// TIA Portal project "PLC_5a_DF_2024compl_V17" (V17)

(* hardware
DEVICE "S7-1200 station_1"  S7-1200 Station
   slot 0: "Telaio di montaggio_0"  S7-1200 Rack  Rack  V1.0
   slot 1: "PLC_ImpiantoCarta"  CPU 1215C DC/DC/Rly  6ES7 215-1HG40-0XB0  V4.5
DEVICE "HMI_1"  TP700 Comfort
   slot 0: "HMI_1"  TP700 Comfort  6AV2 124-0GC01-0AX0  17.0.0.0
   slot 1: "HMI_RT_1"  TP700 Comfort  6AV2 124-0GC01-0AX0  17.0.0.0
   slot 5: "HMI_1.IE_CP_1"  PROFINET Interface  17.0.0.0
      slot 1: "Interfaccia_1 PROFINET"  PROFINET Interface
         slot 1: "Porta_1"  Port
         slot 2: "Porta_2"  Port
   slot 7: "HMI_1.MPI/DP_CP_1"  MPI/DP Interface  17.0.0.0
*)

// ===== PLC "PLC_ImpiantoCarta"  CPU 1215C DC/DC/Rly =====

VAR_GLOBAL   // PLC tag table "Tabella delle variabili standard"
   "M_all_Ms" AT %M10.0 : Bool;   // Memoria allarme Ms
   "M_all_Mn" AT %M10.1 : Bool;   // Memoria allarme Mn
   "M_all_Mp" AT %M10.2 : Bool;   // Memoria allarme Mp
   "M_all_Yv" AT %M10.3 : Bool;   // Memoria allarme Yv
   "Ciclo_Auto" AT %M20.0 : Bool;   // Ciclo automatico
   "Riempimento" AT %M20.1 : Bool;   // Fase 1 di riempimento
   "Caricamento" AT %M20.2 : Bool;   // Fase 2
   "Miscelazione" AT %M20.3 : Bool;   // Fase 3
   "Attesa" AT %M20.4 : Bool;   // Fase 4
   "Svuotamento" AT %M20.5 : Bool;   // Fase 5
   "FN_S4" AT %M40.0 : Bool;   // Fronte discesa S4
   "System_Byte" AT %MB1 : Byte;
   "FirstScan" AT %M1.0 : Bool;
   "DiagStatusUpdate" AT %M1.1 : Bool;
   "AlwaysTRUE" AT %M1.2 : Bool;
   "AlwaysFALSE" AT %M1.3 : Bool;
   "Clock_Byte" AT %MB0 : Byte;
   "Clock_10Hz" AT %M0.0 : Bool;
   "Clock_5Hz" AT %M0.1 : Bool;
   "Clock_2.5Hz" AT %M0.2 : Bool;
   "Clock_2Hz" AT %M0.3 : Bool;
   "Clock_1.25Hz" AT %M0.4 : Bool;
   "Clock_1Hz" AT %M0.5 : Bool;
   "Clock_0.625Hz" AT %M0.6 : Bool;
   "Clock_0.5Hz" AT %M0.7 : Bool;
END_VAR

VAR_GLOBAL   // PLC tag table "IO"
   "S1" AT %I0.0 : Bool;   // Sensore di minimo livello
   "S2" AT %I0.1 : Bool;   // Sensore livello lavoro
   "S3" AT %I0.2 : Bool;   // Sensore di massimo livello
   "S4" AT %I0.3 : Bool;   // Sensore conteggio pezzi
   "Term_Ms" AT %I0.4 : Bool;   // Termico motore Ms (1=OK)
   "Term_Mn" AT %I0.5 : Bool;   // Termico motore Mn (1=OK)
   "Term_Mp" AT %I0.6 : Bool;   // Termico motore Mp (1=OK)
   "YvMicrO" AT %I0.7 : Bool;   // Sensore valvola Yv aperta
   "Motor_Ms" AT %Q0.0 : Bool;   // Motore spappolatore
   "Motor_Mn" AT %Q0.1 : Bool;   // Motore nastro
   "Motor_Mp" AT %Q0.2 : Bool;   // Pompa svuotamento
   "Yv" AT %Q0.3 : Bool;   // Valvola riempimento
   "H1" AT %Q0.4 : Bool;   // Lampada attesa per svuotamento
   "Hs" AT %Q0.5 : Bool;   // Lampada Ms
   "Hn" AT %Q0.6 : Bool;   // Lampada Mn
   "Hp" AT %Q0.7 : Bool;   // Lampada Mp
   "Hv" AT %Q1.0 : Bool;   // Lampada Yv
END_VAR

DATA_BLOCK "DB_HMI"   // DB1
{ S7_Optimized_Access := 'TRUE' }
VERSION : 0.1
   VAR
      SEL_ManAut : Bool;   // SELETTORE DI FUNZIONAMENTO (1=auto)
      Sa : Bool;   // PULSANTE DI START CICLO
      Sp : Bool;   // PULSANTE SVUOTAMENTO
      St : Bool;   // PULSANTE DI STOP CICLO
      Reset : Bool;   // RESET ALLARMI
      CMD_MAN : Struct
         Ms_Start : Bool;   // COMANDO MANUALE START Ms
         Ms_Stop : Bool;   // COMANDO MANUALE ARRESTO Ms
         Mn_Start : Bool;   // COMANDO MANUALE START Mn
         Mn_Stop : Bool;   // COMANDO MANUALE ARRESTO Mn
         Mp_Start : Bool;   // COMANDO MANUALE START Mp
         Mp_Stop : Bool;   // COMANDO MANUALE ARRESTO Mp
         Yv_On : Bool;   // COMANDO MANUALE ECCITA Yv
         Yv_Off : Bool;   // COMANDO MANUALE DISECCITA Yv
      END_STRUCT;
   END_VAR
   VAR RETAIN
      Param : Struct
         PT_Timeout_Yv : Time := T#3s;   // Timeout apertura valvola
         Num_pezzi_da_caricare : Int := 10;   // Numero pezzi da caricare
         Num_pezzi_contati : Int;   // Numero pezzi contati
         Tempo_Miscelazione : Time := T#20S;   // Tempo miscelazione
      END_STRUCT;
   END_VAR
BEGIN
END_DATA_BLOCK

// folder: System blocks/Program resources

DATA_BLOCK "RIT_ALL_Yv"   // DB2
{ S7_Optimized_Access := 'TRUE' }
AUTHOR : Simatic
FAMILY : IEC
NAME : IEC_TMR
VERSION : 1.0
// stored: InstanceOfName IEC_TIMER
"IEC_TIMER"
BEGIN
END_DATA_BLOCK

DATA_BLOCK "DB_Miscelazione"   // DB3
{ S7_Optimized_Access := 'TRUE' }
AUTHOR : Simatic
FAMILY : IEC
NAME : IEC_TMR
VERSION : 1.0
// stored: InstanceOfName IEC_TIMER
"IEC_TIMER"
BEGIN
END_DATA_BLOCK

// folder: (top level)

FUNCTION "DISPOSITIVI" : Void   // FC1, LAD
TITLE = Gestione motori e valvola
{ S7_Optimized_Access := 'TRUE' }
VERSION : 0.1
BEGIN

REGION Network 1: Valvola riempimento
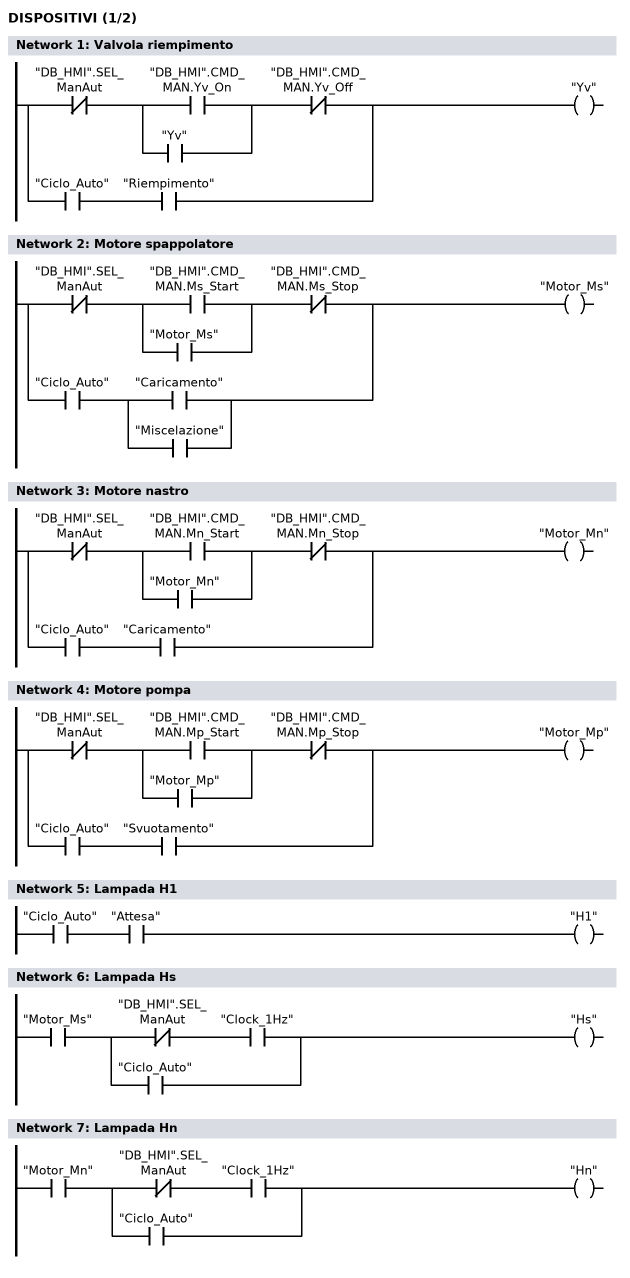
   RUNG wire#powerrail
      I_Contact( "DB_HMI".SEL_ManAut )
      wire#w1
      Contact( "DB_HMI".CMD_MAN.Yv_On )
      wire#w2
      I_Contact( "DB_HMI".CMD_MAN.Yv_Off )
      wire#w3
      Coil( "Yv" )
   END_RUNG
   RUNG wire#w1
      Contact( "Yv" )
   END_RUNG wire#w2
   RUNG wire#powerrail
      Contact( "Ciclo_Auto" )
      Contact( "Riempimento" )
   END_RUNG wire#w3
   // the same network as SCL:
   "Yv" := (NOT "DB_HMI".SEL_ManAut AND ("DB_HMI".CMD_MAN.Yv_On OR "Yv") AND NOT "DB_HMI".CMD_MAN.Yv_Off) OR ("Ciclo_Auto" AND "Riempimento");
END_REGION

REGION Network 2: Motore spappolatore
   RUNG wire#powerrail
      I_Contact( "DB_HMI".SEL_ManAut )
      wire#w1
      Contact( "DB_HMI".CMD_MAN.Ms_Start )
      wire#w2
      I_Contact( "DB_HMI".CMD_MAN.Ms_Stop )
      wire#w3
      Coil( "Motor_Ms" )
   END_RUNG
   RUNG wire#w1
      Contact( "Motor_Ms" )
   END_RUNG wire#w2
   RUNG wire#powerrail
      Contact( "Ciclo_Auto" )
      wire#w4
      Contact( "Caricamento" )
   END_RUNG wire#w3
   RUNG wire#w4
      Contact( "Miscelazione" )
   END_RUNG wire#w3
   // the same network as SCL:
   "Motor_Ms" := (NOT "DB_HMI".SEL_ManAut AND ("DB_HMI".CMD_MAN.Ms_Start OR "Motor_Ms") AND NOT "DB_HMI".CMD_MAN.Ms_Stop) OR ("Ciclo_Auto" AND ("Caricamento" OR "Miscelazione"));
END_REGION

REGION Network 3: Motore nastro
   RUNG wire#powerrail
      I_Contact( "DB_HMI".SEL_ManAut )
      wire#w1
      Contact( "DB_HMI".CMD_MAN.Mn_Start )
      wire#w2
      I_Contact( "DB_HMI".CMD_MAN.Mn_Stop )
      wire#w3
      Coil( "Motor_Mn" )
   END_RUNG
   RUNG wire#w1
      Contact( "Motor_Mn" )
   END_RUNG wire#w2
   RUNG wire#powerrail
      Contact( "Ciclo_Auto" )
      Contact( "Caricamento" )
   END_RUNG wire#w3
   // the same network as SCL:
   "Motor_Mn" := (NOT "DB_HMI".SEL_ManAut AND ("DB_HMI".CMD_MAN.Mn_Start OR "Motor_Mn") AND NOT "DB_HMI".CMD_MAN.Mn_Stop) OR ("Ciclo_Auto" AND "Caricamento");
END_REGION

REGION Network 4: Motore pompa
   RUNG wire#powerrail
      I_Contact( "DB_HMI".SEL_ManAut )
      wire#w1
      Contact( "DB_HMI".CMD_MAN.Mp_Start )
      wire#w2
      I_Contact( "DB_HMI".CMD_MAN.Mp_Stop )
      wire#w3
      Coil( "Motor_Mp" )
   END_RUNG
   RUNG wire#w1
      Contact( "Motor_Mp" )
   END_RUNG wire#w2
   RUNG wire#powerrail
      Contact( "Ciclo_Auto" )
      Contact( "Svuotamento" )
   END_RUNG wire#w3
   // the same network as SCL:
   "Motor_Mp" := (NOT "DB_HMI".SEL_ManAut AND ("DB_HMI".CMD_MAN.Mp_Start OR "Motor_Mp") AND NOT "DB_HMI".CMD_MAN.Mp_Stop) OR ("Ciclo_Auto" AND "Svuotamento");
END_REGION

REGION Network 5: Lampada H1
   RUNG wire#powerrail
      Contact( "Ciclo_Auto" )
      Contact( "Attesa" )
      Coil( "H1" )
   END_RUNG
   // the same network as SCL:
   "H1" := "Ciclo_Auto" AND "Attesa";
END_REGION

REGION Network 6: Lampada Hs
   RUNG wire#powerrail
      Contact( "Motor_Ms" )
      wire#w1
      I_Contact( "DB_HMI".SEL_ManAut )
      Contact( "Clock_1Hz" )
      wire#w2
      Coil( "Hs" )
   END_RUNG
   RUNG wire#w1
      Contact( "Ciclo_Auto" )
   END_RUNG wire#w2
   // the same network as SCL:
   "Hs" := "Motor_Ms" AND ((NOT "DB_HMI".SEL_ManAut AND "Clock_1Hz") OR "Ciclo_Auto");
END_REGION

REGION Network 7: Lampada Hn
   RUNG wire#powerrail
      Contact( "Motor_Mn" )
      wire#w1
      I_Contact( "DB_HMI".SEL_ManAut )
      Contact( "Clock_1Hz" )
      wire#w2
      Coil( "Hn" )
   END_RUNG
   RUNG wire#w1
      Contact( "Ciclo_Auto" )
   END_RUNG wire#w2
   // the same network as SCL:
   "Hn" := "Motor_Mn" AND ((NOT "DB_HMI".SEL_ManAut AND "Clock_1Hz") OR "Ciclo_Auto");
END_REGION

REGION Network 8: Lampada Hp
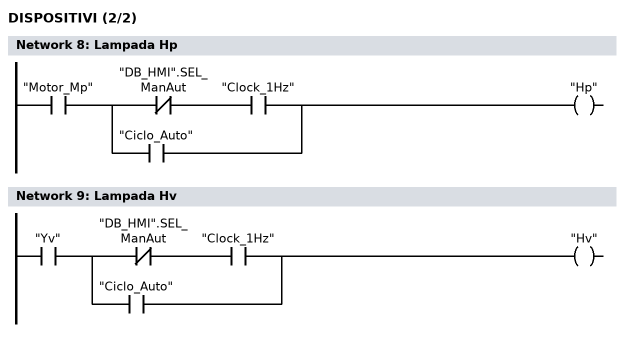
   RUNG wire#powerrail
      Contact( "Motor_Mp" )
      wire#w1
      I_Contact( "DB_HMI".SEL_ManAut )
      Contact( "Clock_1Hz" )
      wire#w2
      Coil( "Hp" )
   END_RUNG
   RUNG wire#w1
      Contact( "Ciclo_Auto" )
   END_RUNG wire#w2
   // the same network as SCL:
   "Hp" := "Motor_Mp" AND ((NOT "DB_HMI".SEL_ManAut AND "Clock_1Hz") OR "Ciclo_Auto");
END_REGION

REGION Network 9: Lampada Hv
   RUNG wire#powerrail
      Contact( "Yv" )
      wire#w1
      I_Contact( "DB_HMI".SEL_ManAut )
      Contact( "Clock_1Hz" )
      wire#w2
      Coil( "Hv" )
   END_RUNG
   RUNG wire#w1
      Contact( "Ciclo_Auto" )
   END_RUNG wire#w2
   // the same network as SCL:
   "Hv" := "Yv" AND ((NOT "DB_HMI".SEL_ManAut AND "Clock_1Hz") OR "Ciclo_Auto");
END_REGION
END_FUNCTION

FUNCTION "ALLARMI" : Void   // FC2, LAD
{ S7_Optimized_Access := 'TRUE' }
VERSION : 0.1
BEGIN

REGION Network 1: ALLARME MOTORE Ms
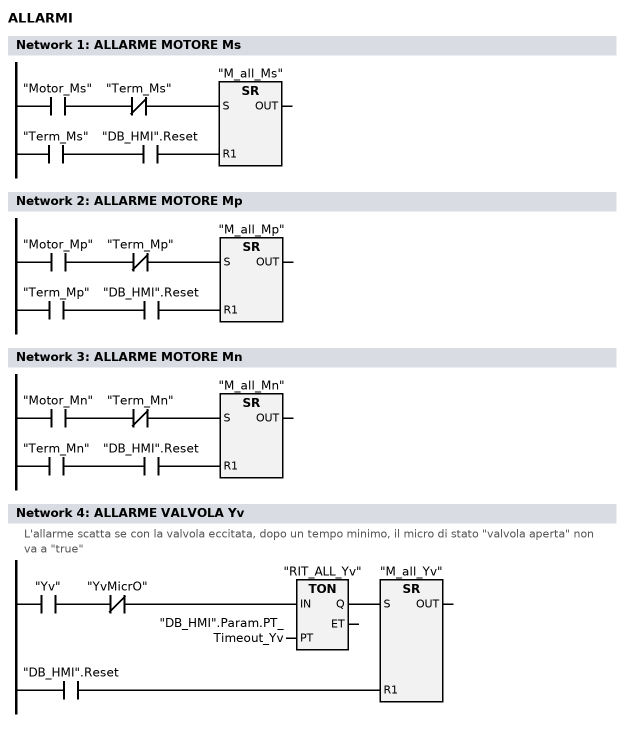
   RUNG wire#powerrail
      Contact( "Motor_Ms" )
      I_Contact( "Term_Ms" )
      S_SR(operand := "M_all_Ms", r1 := wire#w1)
   END_RUNG
   RUNG wire#powerrail
      Contact( "Term_Ms" )
      Contact( "DB_HMI".Reset )
   END_RUNG wire#w1
   // the same network as SCL:
   IF "Motor_Ms" AND NOT "Term_Ms" THEN
       "M_all_Ms" := TRUE;   // SR flip-flop
   END_IF;
   IF "Term_Ms" AND "DB_HMI".Reset THEN "M_all_Ms" := FALSE; END_IF;
END_REGION

REGION Network 2: ALLARME MOTORE Mp
   RUNG wire#powerrail
      Contact( "Motor_Mp" )
      I_Contact( "Term_Mp" )
      S_SR(operand := "M_all_Mp", r1 := wire#w1)
   END_RUNG
   RUNG wire#powerrail
      Contact( "Term_Mp" )
      Contact( "DB_HMI".Reset )
   END_RUNG wire#w1
   // the same network as SCL:
   IF "Motor_Mp" AND NOT "Term_Mp" THEN
       "M_all_Mp" := TRUE;   // SR flip-flop
   END_IF;
   IF "Term_Mp" AND "DB_HMI".Reset THEN "M_all_Mp" := FALSE; END_IF;
END_REGION

REGION Network 3: ALLARME MOTORE Mn
   RUNG wire#powerrail
      Contact( "Motor_Mn" )
      I_Contact( "Term_Mn" )
      S_SR(operand := "M_all_Mn", r1 := wire#w1)
   END_RUNG
   RUNG wire#powerrail
      Contact( "Term_Mn" )
      Contact( "DB_HMI".Reset )
   END_RUNG wire#w1
   // the same network as SCL:
   IF "Motor_Mn" AND NOT "Term_Mn" THEN
       "M_all_Mn" := TRUE;   // SR flip-flop
   END_IF;
   IF "Term_Mn" AND "DB_HMI".Reset THEN "M_all_Mn" := FALSE; END_IF;
END_REGION

REGION Network 4: ALLARME VALVOLA Yv
   // L'allarme scatta se con la valvola eccitata, dopo un tempo minimo, il micro di stato "valvola aperta" non va a "true"
   "RIT_ALL_Yv".TON(IN := "Yv" AND NOT "YvMicrO", PT := "DB_HMI".Param.PT_Timeout_Yv);
   IF "RIT_ALL_Yv".Q THEN
       "M_all_Yv" := TRUE;   // SR flip-flop
   END_IF;
   IF "DB_HMI".Reset THEN "M_all_Yv" := FALSE; END_IF;
END_REGION
END_FUNCTION

FUNCTION "CICLO_AUTOMATICO" : Void   // FC3, LAD
{ S7_Optimized_Access := 'TRUE' }
VERSION : 0.1
   VAR_TEMP   // added for the SCL form of the ladder/FBD networks
      _w1 : Bool;
   END_VAR
BEGIN

REGION Network 1: STOP CICLO (MOMENTANEO)
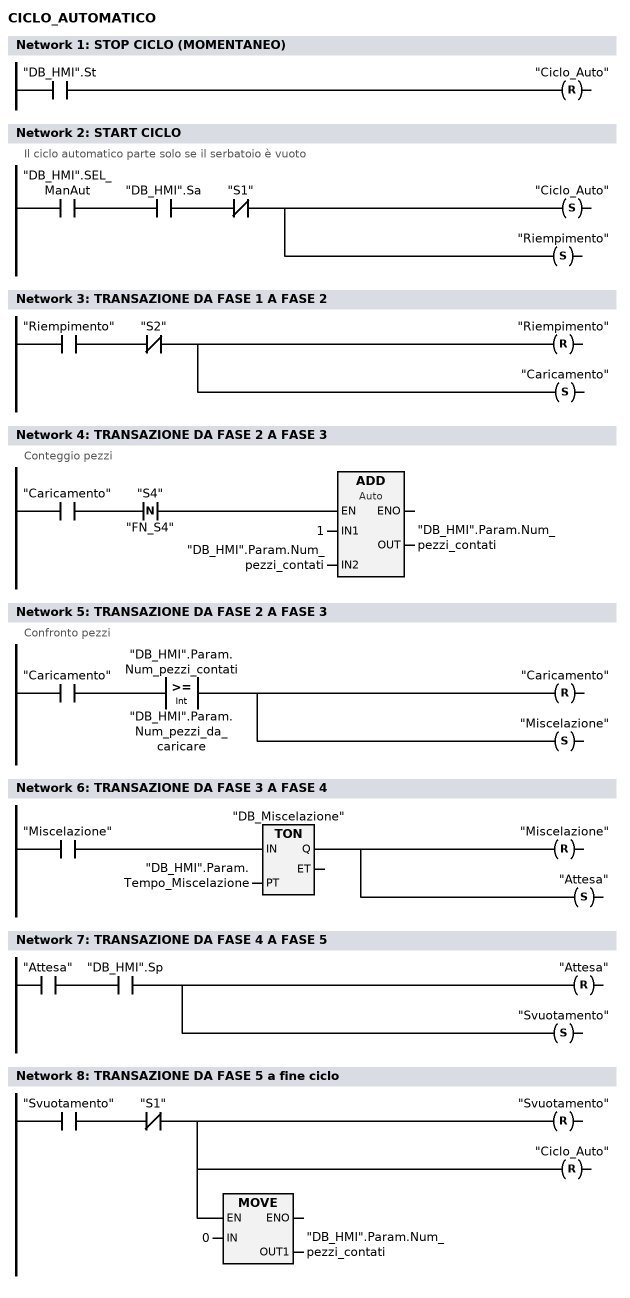
   RUNG wire#powerrail
      Contact( "DB_HMI".St )
      R_Coil( "Ciclo_Auto" )
   END_RUNG
   // the same network as SCL:
   IF "DB_HMI".St THEN "Ciclo_Auto" := FALSE; END_IF;
END_REGION

REGION Network 2: START CICLO
   // Il ciclo automatico parte solo se il serbatoio è vuoto
   RUNG wire#powerrail
      Contact( "DB_HMI".SEL_ManAut )
      Contact( "DB_HMI".Sa )
      I_Contact( "S1" )
      wire#w1
      S_Coil( "Ciclo_Auto" )
   END_RUNG
   RUNG wire#w1
      S_Coil( "Riempimento" )
   END_RUNG
   // the same network as SCL:
   IF "DB_HMI".SEL_ManAut AND "DB_HMI".Sa AND NOT "S1" THEN
       "Ciclo_Auto" := TRUE;
       "Riempimento" := TRUE;
   END_IF;
END_REGION

REGION Network 3: TRANSAZIONE DA FASE 1 A FASE 2
   RUNG wire#powerrail
      Contact( "Riempimento" )
      I_Contact( "S2" )
      wire#w1
      R_Coil( "Riempimento" )
   END_RUNG
   RUNG wire#w1
      S_Coil( "Caricamento" )
   END_RUNG
   // the same network as SCL:
   #_w1 := "Riempimento" AND NOT "S2";
   IF #_w1 THEN
       "Riempimento" := FALSE;
       "Caricamento" := TRUE;
   END_IF;
END_REGION

REGION Network 4: TRANSAZIONE DA FASE 2 A FASE 3
   // Conteggio pezzi
   RUNG wire#powerrail
      Contact( "Caricamento" )
      N_Contact(operand := "S4", bit := "FN_S4")
      Add(in1 := 1, in2 := "DB_HMI".Param.Num_pezzi_contati, out => "DB_HMI".Param.Num_pezzi_contati)
   END_RUNG
   // the same network as SCL:
   #_w1 := "Caricamento" AND NOT "S4" AND "FN_S4";   // falling edge of "S4"
   "FN_S4" := "S4";
   IF #_w1 THEN "DB_HMI".Param.Num_pezzi_contati := 1 + "DB_HMI".Param.Num_pezzi_contati; END_IF;
END_REGION

REGION Network 5: TRANSAZIONE DA FASE 2 A FASE 3
   // Confronto pezzi
   RUNG wire#powerrail
      Contact( "Caricamento" )
      { S7_Templates := "SrcType := Int" } GE_Contact(in1 := "DB_HMI".Param.Num_pezzi_contati, in2 := "DB_HMI".Param.Num_pezzi_da_caricare)
      wire#w1
      R_Coil( "Caricamento" )
   END_RUNG
   RUNG wire#w1
      S_Coil( "Miscelazione" )
   END_RUNG
   // the same network as SCL:
   #_w1 := "Caricamento" AND ("DB_HMI".Param.Num_pezzi_contati >= "DB_HMI".Param.Num_pezzi_da_caricare);
   IF #_w1 THEN
       "Caricamento" := FALSE;
       "Miscelazione" := TRUE;
   END_IF;
END_REGION

REGION Network 6: TRANSAZIONE DA FASE 3 A FASE 4
   "DB_Miscelazione".TON(IN := "Miscelazione", PT := "DB_HMI".Param.Tempo_Miscelazione);
   IF "DB_Miscelazione".Q THEN
       "Miscelazione" := FALSE;
       "Attesa" := TRUE;
   END_IF;
END_REGION

REGION Network 7: TRANSAZIONE DA FASE 4 A FASE 5
   RUNG wire#powerrail
      Contact( "Attesa" )
      Contact( "DB_HMI".Sp )
      wire#w1
      R_Coil( "Attesa" )
   END_RUNG
   RUNG wire#w1
      S_Coil( "Svuotamento" )
   END_RUNG
   // the same network as SCL:
   #_w1 := "Attesa" AND "DB_HMI".Sp;
   IF #_w1 THEN
       "Attesa" := FALSE;
       "Svuotamento" := TRUE;
   END_IF;
END_REGION

REGION Network 8: TRANSAZIONE DA FASE 5 a fine ciclo
   RUNG wire#powerrail
      Contact( "Svuotamento" )
      I_Contact( "S1" )
      wire#w1
      R_Coil( "Svuotamento" )
   END_RUNG
   RUNG wire#w1
      R_Coil( "Ciclo_Auto" )
   END_RUNG
   RUNG wire#w1
      Move(in := 0, out1 => "DB_HMI".Param.Num_pezzi_contati)
   END_RUNG
   // the same network as SCL:
   #_w1 := "Svuotamento" AND NOT "S1";
   IF #_w1 THEN
       "Svuotamento" := FALSE;
       "Ciclo_Auto" := FALSE;
       "DB_HMI".Param.Num_pezzi_contati := 0;
   END_IF;
END_REGION
END_FUNCTION

ORGANIZATION_BLOCK "Main"   // OB1, LAD, ProgramCycle
TITLE = "Main Program Sweep (Cycle)"
{ S7_Optimized_Access := 'TRUE' }
VERSION : 0.1
   VAR_INPUT
      Initial_Call : Bool;   // Initial call of this OB
      Remanence : Bool;   // =True, if remanent data are available
   END_VAR
BEGIN

REGION Network 1
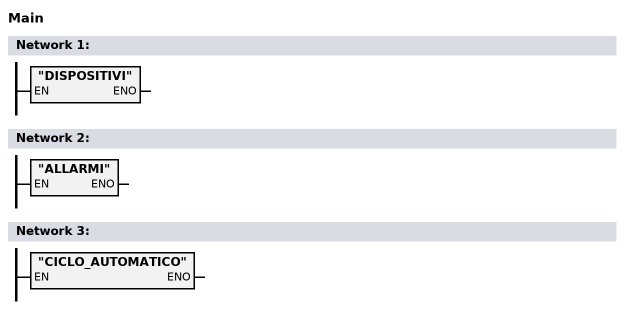
   RUNG wire#powerrail
      "DISPOSITIVI"()
   END_RUNG
   // the same network as SCL:
   "DISPOSITIVI"();
END_REGION

REGION Network 2
   RUNG wire#powerrail
      "ALLARMI"()
   END_RUNG
   // the same network as SCL:
   "ALLARMI"();
END_REGION

REGION Network 3
   RUNG wire#powerrail
      "CICLO_AUTOMATICO"()
   END_RUNG
   // the same network as SCL:
   "CICLO_AUTOMATICO"();
END_REGION
END_ORGANIZATION_BLOCK

(* ===== HMI "HMI_RT_1" =====
system functions are stored by id; their names below are inferred from use
connection "HMI_Collegamento_2": ETHERNET, S7_1200_OMS

HMI tags "Tabella delle variabili standard"
   "S3" : Bool = PLC S3 AT %I0.2, 1 s
   "Ms" : Bool = PLC Motor_Ms AT %Q0.0, 1 s
   "Mp" : Bool = PLC Motor_Mp AT %Q0.2, 1 s
   "Mn" : Bool = PLC Motor_Mn AT %Q0.1, 1 s
   "S4" : Bool = PLC S4 AT %I0.3, 1 s
   "S1" : Bool = PLC S1 AT %I0.0, 1 s
   "S2" : Bool = PLC S2 AT %I0.1, 1 s
   "Ciclo_Auto" : Bool = PLC Ciclo_Auto AT %M20.0, 1 s
   "Sa" : Bool = PLC DB_HMI.Sa AT %I0.0, 1 s
   "DB_HMI_CMD_MAN_Mn_Start" : Bool = PLC DB_HMI.CMD_MAN.Mn_Start, 1 s
   "DB_HMI_CMD_MAN_Mn_Stop" : Bool = PLC DB_HMI.CMD_MAN.Mn_Stop, 1 s
   "DB_HMI_Sp" : Bool = PLC DB_HMI.Sp, 1 s
   "DB_HMI_Sa" : Bool = PLC DB_HMI.Sa, 1 s
   "DB_HMI_SEL_ManAut" : Bool = PLC DB_HMI.SEL_ManAut, 1 s
   "DB_HMI_CMD_MAN_Mp_Start" : Bool = PLC DB_HMI.CMD_MAN.Mp_Start, 1 s
   "DB_HMI_CMD_MAN_Mp_Stop" : Bool = PLC DB_HMI.CMD_MAN.Mp_Stop, 1 s
   "DB_HMI_CMD_MAN_Ms_Start" : Bool = PLC DB_HMI.CMD_MAN.Ms_Start, 1 s
   "DB_HMI_CMD_MAN_Ms_Stop" : Bool = PLC DB_HMI.CMD_MAN.Ms_Stop, 1 s
   "DB_HMI_CMD_MAN_Yv_on" : Bool = PLC DB_HMI.CMD_MAN.Yv_On, 1 s
   "DB_HMI_CMD_MAN_Yv_off" : Bool = PLC DB_HMI.CMD_MAN.Yv_Off, 1 s
   "Yv" : Bool = PLC Yv AT %Q0.3, 1 s
   "SEL" : Bool = PLC DB_HMI.SEL_ManAut AT %I0.0, 1 s
   "Hv" : Bool = PLC Hv AT %Q1.0, 1 s
   "Hn" : Bool = PLC Hn AT %Q0.6, 1 s
   "Hs" : Bool = PLC Hs AT %Q0.5, 1 s
   "Hp" : Bool = PLC Hp AT %Q0.7, 1 s
   "DB_HMI_Param_Num_pezzi_da_caricare" : Int = PLC DB_HMI.Param.Num_pezzi_contati, 1 s
   "DB_HMI_Param_Num_pezzi_contati" : Int = PLC DB_HMI.Param.Num_pezzi_da_caricare, 1 s
   "DB_HMI_Param_Tempo_Miscelazione" : Time = PLC DB_HMI.Param.Tempo_Miscelazione, 1 s
   "DB_HMI_Reset" : Bool = PLC DB_HMI.Reset, 1 s
   "DB_HMI_St" : Bool = PLC DB_HMI.St, 1 s
   "Miscelazione" : Bool = PLC Miscelazione AT %M20.3, 1 s

HMI tags "ALARMS"
   "Alarms" : Word AT %MW10, 1 s

discrete alarms
   1: '00.00', class Errors, trigger "Alarms" bit 0
   2: '00.01', class Errors, trigger "Alarms" bit 1
   3: '00.02', class Errors, trigger "Alarms" bit 2
   4: '00.03', class Errors, trigger "Alarms" bit 3
   5: '00.04', class Errors, trigger "Alarms" bit 4
   6: '00.05', class Errors, trigger "Alarms" bit 5
   7: '00.06', class Errors, trigger "Alarms" bit 6
   8: '00.07', class Errors, trigger "Alarms" bit 7
   9: '00.08 Memoria allarme Ms', class Errors, trigger "Alarms" bit 8
   10: '00.09 Memoria allarme Mn', class Errors, trigger "Alarms" bit 9
   11: '00.10 Memoria allarme Mp', class Errors, trigger "Alarms" bit 10
   12: '00.11 Memoria allarme Yv', class Errors, trigger "Alarms" bit 11
   13: '00.12', class Errors, trigger "Alarms" bit 12
   14: '00.13', class Errors, trigger "Alarms" bit 13
   15: '00.14', class Errors, trigger "Alarms" bit 14
   16: '00.15', class Errors, trigger "Alarms" bit 15

screen "01 Main" 800x480
   GraphicView "Vista grafica_1" at 0,0 size 799x479; Picture "logoitis_arancio"
   Button "Pulsante_1" at 0,0 size 798x425; TextOff 'Text'
      on Click: ActivateScreen("02 Sinottico", 0)
   TextField "Casella di testo_1" at 446,431 size 323x28; Text 'Operatore: Isabel Rodolico / OPERATORE :Isabel Rodolico'
   Button "Pulsante_5" at 0,441 size 96x38; TextOff 'ALLARMI'; PictureOff "NavigateHome_KTP400_Comfort_TR"
      on Click: ActivateScreen("100 ALLARMI", 0)
      Appearance <- "Alarms"

screen "02 Sinottico" 800x480
   Button "Pulsante_1" at 703,441 size 96x38; TextOff 'Text'; PictureOff "Right_Arrow_1"
      on Click: ActivateScreen("03 Parametri produzione", 0)
   Button "Pulsante_3" at 0,442 size 96x38; TextOff 'Text'; PictureOff "NavigateHome_KTP400_Comfort_TR"
      on Click: ActivateScreen("01 Main", 0)
   Switch "Interruttore_1" at 503,77 size 141x53; TextOn 'MAN. / AUTO'; CaptionText 'CICLO / AVVIO'; TextOff 'AUTO / MAN'; Authorization "operazione"
      ProcessValue <- "DB_HMI_SEL_ManAut"
   Button "Pulsante_4" at 704,441 size 96x39; TextOff 'Text'; PictureOff "Right_Arrow_1"
      on Click: ActivateScreen("03 Parametri produzione", 0)
   GraphicView "Vista grafica_9" at 306,127 size 463x267; Picture "Grafica_10"
   GraphicView "Vista grafica_1" at 200,161 size 158x198; Picture "Grafica_30"
   GraphicView "Vista grafica_2" at 234,351 size 30x32; Picture "Grafica_28"
   GraphicView "Vista grafica_3" at 98,361 size 145x27; Picture "Grafica_29"
   GraphicView "Vista grafica_7" at 45,366 size 61x45; Picture "Grafica_34"
   Group "Group_S2" at 141,235 size 38x23
   Group "Group_S3" at 141,206 size 38x23
   Group "Group_S4" at 301,102 size 38x23
   Group "Group_S1" at 374,292 size 38x23
   Circle "S3" at 201,205 size 16x16
      Appearance <- "S3"
   Circle "S2" at 202,236 size 16x16
      Appearance <- "S2"
   GraphicView "Vista grafica_8" at 231,322 size 92x25; Picture "Grafica_35"
   Circle "lampadaHpMan" at 161,367 size 16x16
      Visibility <- "DB_HMI_SEL_ManAut"
      Appearance <- "Hp"
   Circle "S1" at 343,292 size 16x16
      Appearance <- "S1"
   Circle "S4" at 311,137 size 16x16
      Appearance <- "S4"
   Circle "lampadaHnMan" at 742,375 size 16x16
      Visibility <- "DB_HMI_SEL_ManAut"
      Appearance <- "Hn"
   Circle "lampadaHsMan" at 270,327 size 16x16
      Visibility <- "DB_HMI_SEL_ManAut"
      Appearance <- "Hs"
   Group "Group_1" at 27,133 size 241x29; Picture "Grafica_33"
   Button "Pulsante_10" at 677,141 size 80x50; TextOff 'STOP'
      on Release: ResetBit("DB_HMI_St")
      on Press: SetBit("DB_HMI_St")
   Button "Pulsante_11" at 677,77 size 80x50; TextOff 'START'
      on Release: ResetBit("DB_HMI_Sa")
      on Press: SetBit("DB_HMI_Sa")
   Circle "lampadaYvMan" at 161,136 size 16x16
      Visibility <- "DB_HMI_SEL_ManAut"
      Appearance <- "Hv"
   Button "Pulsante_2" at 677,209 size 80x50; TextOff 'STOP / SVUOTA'
      on Release: ResetBit("DB_HMI_Sp")
      on Press: SetBit("DB_HMI_Sp")
   Button "Pulsante_5" at 0,0 size 96x38; TextOff 'ALLARMI'; PictureOff "NavigateHome_KTP400_Comfort_TR"
      on Click: ActivateScreen("100 ALLARMI", 0)
      Appearance <- "Alarms"
   TextField "Casella di testo_8" at 300,0 size 165x34; Text 'SINOTTICO / SONOTTICO'
   Rectangle "Rettangolo_11" at 670,64 size 97x199
      Visibility <- "DB_HMI_SEL_ManAut"
   Rectangle "Rettangolo_1" at 150,92 size 38x18
      Appearance <- "Hv"
   TextField "Casella di testo_1" at 156,90 size 27x23; Text 'Yv'
   Rectangle "Rettangolo_2" at 264,362 size 38x18
      Appearance <- "Hs"
   TextField "Ms" at 270,360 size 29x23; Text 'Ms'
   TextField "Casella di testo_3" at 147,235 size 27x23; Text 'S2'
   TextField "Casella di testo_4" at 147,206 size 27x23; Text 'S3'
   TextField "Casella di testo_5" at 307,102 size 27x23; Text 'S4'
   TextField "Casella di testo_6" at 380,292 size 27x23; Text 'S1'
   Rectangle "Rettangolo_8" at 731,406 size 38x18
      Appearance <- "Hn"
   TextField "Casella di testo_7" at 737,404 size 31x23; Text 'Mn'
   GraphicView "Vista grafica_6" at 152,137 size 36x16; Picture "Grafica_33"
   GraphicView "Vista grafica_4" at 238,137 size 30x25; Picture "Grafica_32"
   GraphicView "Vista grafica_5" at 27,133 size 221x22; Picture "Grafica_29"
   Button "Pulsante_MN" at 730,399 size 44x32; TextOff 'Text'
      on Click: function_efd93a16("Pagina popupMn", 420, 20, -1, -1, 1)
      Visibility <- "DB_HMI_SEL_ManAut"
   Button "Pulsante_MP" at 149,326 size 44x32; TextOff 'Text'
      on Click: function_efd93a16("Pagina popupMp", 420, 20, -1, -1, 1)
      Visibility <- "DB_HMI_SEL_ManAut"
   Button "Pulsante_YV" at 149,85 size 44x32; TextOff 'Text'
      on Click: function_efd93a16("Pagina popupYv", 420, 20, -1, -1, 1)
      Visibility <- "DB_HMI_SEL_ManAut"
   Button "Pulsante_MS" at 263,356 size 44x32; TextOff 'Text'
      on Click: function_efd93a16("Pagina popupMs", 420, 20, -1, -1, 1)
      Visibility <- "DB_HMI_SEL_ManAut"
   GraphicView "Vista grafica_14" at 564,113 size 15x24; Picture "Lucchetto"
      Visibility <- "DB_HMI_SEL_ManAut"
   Group "Group_Ms" at 264,360 size 38x23
   Group "Group_Mn" at 731,404 size 38x23
   Group "GroupYv" at 150,90 size 38x23
   Group "GroupMp" at 150,333 size 38x23
   Rectangle "Rettangolo_3" at 150,335 size 38x18
      Appearance <- "Hp"
   TextField "Casella di testo_2" at 156,333 size 31x23; Text 'Yv / Mp'

screen "100 ALLARMI" 800x480
   AlarmView "Vista segnalazioni_1" at 0,37 size 799x398
   Button "Pulsante_3" at 0,432 size 96x47; TextOff 'Text'; PictureOff "NavigateHome_KTP400_Comfort_TR"
      on Click: ActivateScreen("01 Main", 0)
   TextField "Casella di testo_1" at 339,3 size 122x33; Text 'ALLARMI'
   Button "Pulsante_1" at 97,432 size 623x47; TextOff 'RESET'
      on Press: function_b14e0dd5("DB_HMI_Reset", 0)

screen "03 Parametri produzione" 800x480
   Button "Pulsante_4" at 704,442 size 96x38; TextOff 'Text'; PictureOff "Right_Arrow_1"
      on Click: ActivateScreen("01 Main", 0)
   Button "Pulsante_2" at 0,442 size 96x38; TextOff 'Text'; PictureOff "Left_Arrow_1"
      on Click: ActivateScreen("02 Sinottico", 0)
   IOField "Campo I/O_2" at 698,193 size 102x50; FormatPattern s999
      Appearance <- "Ciclo_Auto"
      ProcessValue <- "DB_HMI_Param_Num_pezzi_contati"
      ObjectEnable <- "Ciclo_Auto"
   IOField "Campo I/O_3" at 698,289 size 102x50; Authorization "amministrazione"; FormatPattern 999
      ObjectEnable <- "Ciclo_Auto"
      Appearance <- "Ciclo_Auto"
      ProcessValue <- "Miscelazione"
   TextField "Casella di testo_2" at 9,104 size 364x34; Text 'PANI IN CARICAMENTO / PANI TOTALI DA VERSARE'
   TextField "Casella di testo_3" at 10,200 size 354x34; Text 'PANI CARICATI / PANI EFFETTIVI VERSATI'
   TextField "Casella di testo_4" at 10,296 size 352x34; Text 'DURATA MISCELAZIONE / TEMPO DI MISCELAZIONE'
   IOField "Campo I/O_1" at 698,97 size 102x50; Authorization "amministrazione"; FormatPattern s999
      ProcessValue <- "DB_HMI_Param_Num_pezzi_da_caricare"
   TextField "Casella di testo_8" at 223,0 size 402x34; Text 'SINOTTICO / PARAMETRI DI PRODUZIONE'
   Button "Pulsante_5" at 0,0 size 96x40; TextOff 'ALLARMI'; PictureOff "NavigateHome_KTP400_Comfort_TR"
      on Click: ActivateScreen("100 ALLARMI", 0)
      Appearance <- "Alarms"
   TextField "Casella di testo_1" at 300,0 size 186x34; Text 'PRODUZIONE'
   GraphicView "Vista grafica_14" at 772,126 size 15x24; Picture "Lucchetto"
      Visibility <- "DB_HMI_SEL_ManAut"
   GraphicView "Vista grafica_1" at 772,315 size 15x24; Picture "Lucchetto"
      Visibility <- "DB_HMI_SEL_ManAut"

Template "TEM" 800x480
   Button "Pulsante_5" at 0,1 size 96x38; TextOff 'ALLARMI'; PictureOff "NavigateHome_KTP400_Comfort_TR"
      on Click: ActivateScreen("100 ALLARMI", 0)

PopupScreen "Pagina popupMs" 350x180
   Button "Pulsante_1" at 29,85 size 95x43; TextOff 'START'
      on Release: ResetBit("DB_HMI_CMD_MAN_Ms_Start")
      on Press: SetBit("DB_HMI_CMD_MAN_Ms_Start")
   Button "Pulsante_3" at 199,85 size 95x43; TextOff 'STOP'
      on Release: ResetBit("DB_HMI_CMD_MAN_Ms_Stop")
      on Press: SetBit("DB_HMI_CMD_MAN_Ms_Stop")
   TextField "Casella di testo_1" at 76,26 size 212x21; Text 'ABILITAZIONE MANUALE SPAPPOLATORE / ABILITAZIONE MANUALE'
   TextField "Casella di testo_2" at 104,47 size 131x21; Text 'ABILITAZIONE MANUALE SPAPPOLATORE / SPAPPOLATORE'
   Button "Pulsante_2" at 322,0 size 25x26; TextOff 'Text'; PictureOff "ExitRuntime_KTP400_Comfort_TR"
      on Click: ActivateScreen("02 Sinottico", 0)

PopupScreen "Pagina popupMp" 350x180
   Button "Pulsante_2" at 325,0 size 25x26; TextOff 'Text'; PictureOff "ExitRuntime_KTP400_Comfort_TR"
      on Click: ActivateScreen("02 Sinottico", 0)
   Button "Pulsante_1" at 29,85 size 95x43; TextOff 'START'
      on Release: ResetBit("DB_HMI_CMD_MAN_Mp_Start")
      on Press: SetBit("DB_HMI_CMD_MAN_Mp_Start")
   Button "Pulsante_3" at 199,85 size 95x43; TextOff 'STOP'
      on Release: ResetBit("DB_HMI_CMD_MAN_Mp_Stop")
      on Press: SetBit("DB_HMI_CMD_MAN_Mp_Stop")
   TextField "Casella di testo_1" at 32,36 size 268x21; Text 'ABILITAZIONE MANUALE POMPA'

PopupScreen "Pagina popupMn" 350x180
   Button "Pulsante_2" at 325,0 size 25x26; TextOff 'Text'; PictureOff "ExitRuntime_KTP400_Comfort_TR"
      on Click: ActivateScreen("02 Sinottico", 0)
   Button "Pulsante_1" at 29,85 size 95x43; TextOff 'START'
      on Release: ResetBit("DB_HMI_CMD_MAN_Mn_Start")
      on Press: SetBit("DB_HMI_CMD_MAN_Mn_Start")
   Button "Pulsante_3" at 199,85 size 95x43; TextOff 'STOP'
      on Release: ResetBit("DB_HMI_CMD_MAN_Mn_Stop")
      on Press: SetBit("DB_HMI_CMD_MAN_Mn_Stop")
   TextField "Casella di testo_1" at 32,36 size 278x21; Text 'ABILITAZIONE MANUALE NASTRO'

PopupScreen "Pagina popupYv" 350x180
   Button "Pulsante_2" at 325,0 size 25x26; TextOff 'Text'; PictureOff "ExitRuntime_KTP400_Comfort_TR"
      on Click: ActivateScreen("02 Sinottico", 0)
   Button "Pulsante_1" at 29,85 size 95x43; TextOff 'START'
      on Release: ResetBit("DB_HMI_CMD_MAN_Yv_on")
      on Press: SetBit("DB_HMI_CMD_MAN_Yv_on")
   Button "Pulsante_3" at 199,85 size 95x43; TextOff 'STOP'
      on Release: ResetBit("DB_HMI_CMD_MAN_Yv_off")
      on Press: SetBit("DB_HMI_CMD_MAN_Yv_off")
   TextField "Casella di testo_1" at 32,36 size 286x21; Text 'ABILITAZIONE MANUALE VALVOLA'
*)